FUNCTION_BLOCK TaurusLed 
VAR
	_text : T_MaxString;

	
END_VAR

PROPERTY Text : STRING
GET
Text := _text;
END_GET
SET
_text := Text;
END_SET
END_PROPERTY

END_FUNCTION_BLOCK

(* stored: Version 1.1.0.1, ProductVersion 3.1.4024.12
   POU TaurusLed: Id {e63cee5b-d7be-43fb-a377-2aa3bbe5386e}, SpecialFunc None
   Property Text: Id {b753cbdf-f104-4e01-8e2f-6f6d5bb31d2f}
   Get Get: Id {bed5069e-410c-4790-bead-a7d8591095b0}
   Set Set: Id {e42b9ef2-96ee-452e-9dd0-944c0239a58f} *)
